// TIA Portal V18 export
// export: Created 2026-06-08T16:32:21.3339851Z, ExportSetting WithDefaults, DisplayName Totally Integrated Automation Portal, DisplayVersion V18, DisplayName TIA Portal Openness, DisplayVersion V18, DisplayName TIA Portal Version Control Interface, DisplayVersion V18, DisplayName STEP 7 Professional, DisplayVersion V18, DisplayName STEP 7 Safety, DisplayVersion V18, DisplayName WinCC Professional, DisplayVersion V18
FUNCTION_BLOCK "Assembly_conv"   // FB9, LAD
VERSION : 0.1
// stored: AutoNumber true, IsIECCheckEnabled false, UDAEnableTagReadback false
   VAR_TEMP   // added for the SCL form of the ladder/FBD networks
      _w1 : Bool;
      _s5time1 : S5Time;
   END_VAR
BEGIN

REGION Network 1
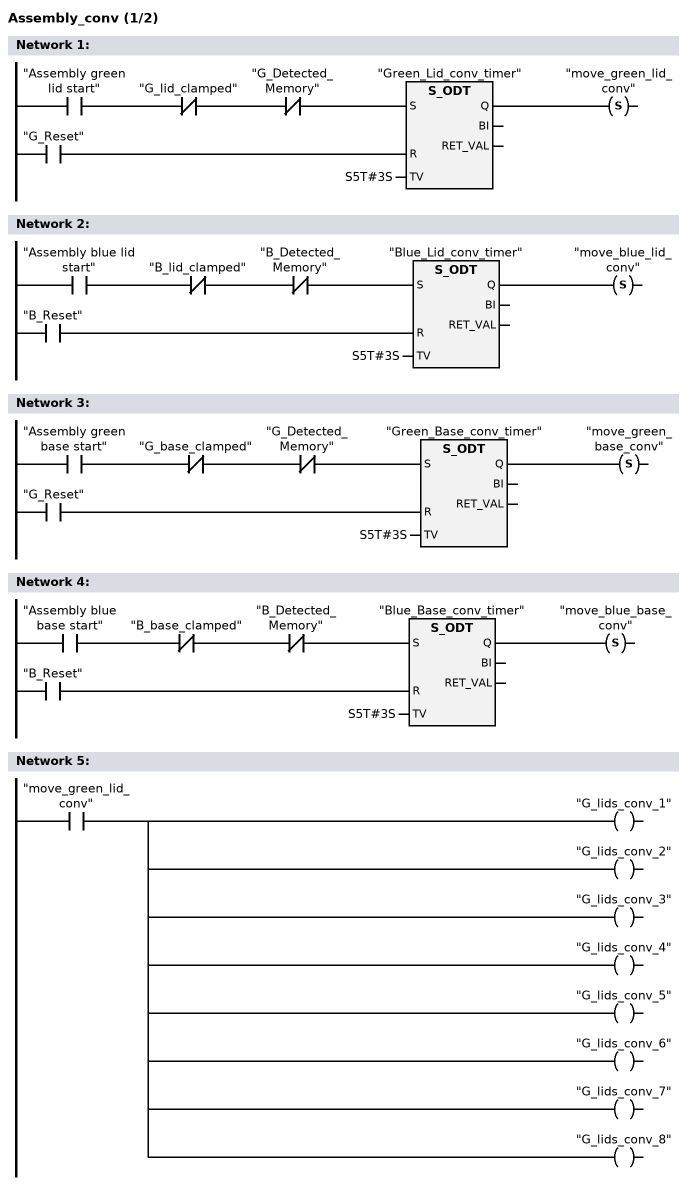
   RUNG wire#powerrail
      Contact( "Assembly green lid start" )
      I_Contact( "G_lid_clamped" )
      I_Contact( "G_Detected_Memory" )
      S_ODT(T_NO := "Green_Lid_conv_timer", R := wire#w1, TV := S5T#3S, BI =>, RET_VAL =>)
      S_Coil( "move_green_lid_conv" )
   END_RUNG
   RUNG wire#powerrail
      Contact( "G_Reset" )
   END_RUNG wire#w1
   // the same network as SCL:
   #_s5time1 := S_ODT(T_NO := "Green_Lid_conv_timer",
                      S := "Assembly green lid start" AND NOT "G_lid_clamped" AND NOT "G_Detected_Memory",
                      R := "G_Reset",
                      TV := S5T#3S,
                      Q => #_w1);
   IF #_w1 THEN "move_green_lid_conv" := TRUE; END_IF;
END_REGION

REGION Network 2
   RUNG wire#powerrail
      Contact( "Assembly blue lid start" )
      I_Contact( "B_lid_clamped" )
      I_Contact( "B_Detected_Memory" )
      S_ODT(T_NO := "Blue_Lid_conv_timer", R := wire#w1, TV := S5T#3S, BI =>, RET_VAL =>)
      S_Coil( "move_blue_lid_conv" )
   END_RUNG
   RUNG wire#powerrail
      Contact( "B_Reset" )
   END_RUNG wire#w1
   // the same network as SCL:
   #_s5time1 := S_ODT(T_NO := "Blue_Lid_conv_timer",
                      S := "Assembly blue lid start" AND NOT "B_lid_clamped" AND NOT "B_Detected_Memory",
                      R := "B_Reset",
                      TV := S5T#3S,
                      Q => #_w1);
   IF #_w1 THEN "move_blue_lid_conv" := TRUE; END_IF;
END_REGION

REGION Network 3
   RUNG wire#powerrail
      Contact( "Assembly green base start" )
      I_Contact( "G_base_clamped" )
      I_Contact( "G_Detected_Memory" )
      S_ODT(T_NO := "Green_Base_conv_timer", R := wire#w1, TV := S5T#3S, BI =>, RET_VAL =>)
      S_Coil( "move_green_base_conv" )
   END_RUNG
   RUNG wire#powerrail
      Contact( "G_Reset" )
   END_RUNG wire#w1
   // the same network as SCL:
   #_s5time1 := S_ODT(T_NO := "Green_Base_conv_timer",
                      S := "Assembly green base start" AND NOT "G_base_clamped" AND NOT "G_Detected_Memory",
                      R := "G_Reset",
                      TV := S5T#3S,
                      Q => #_w1);
   IF #_w1 THEN "move_green_base_conv" := TRUE; END_IF;
END_REGION

REGION Network 4
   RUNG wire#powerrail
      Contact( "Assembly blue base start" )
      I_Contact( "B_base_clamped" )
      I_Contact( "B_Detected_Memory" )
      S_ODT(T_NO := "Blue_Base_conv_timer", R := wire#w1, TV := S5T#3S, BI =>, RET_VAL =>)
      S_Coil( "move_blue_base_conv" )
   END_RUNG
   RUNG wire#powerrail
      Contact( "B_Reset" )
   END_RUNG wire#w1
   // the same network as SCL:
   #_s5time1 := S_ODT(T_NO := "Blue_Base_conv_timer",
                      S := "Assembly blue base start" AND NOT "B_base_clamped" AND NOT "B_Detected_Memory",
                      R := "B_Reset",
                      TV := S5T#3S,
                      Q => #_w1);
   IF #_w1 THEN "move_blue_base_conv" := TRUE; END_IF;
END_REGION

REGION Network 5
   RUNG wire#powerrail
      Contact( "move_green_lid_conv" )
      wire#w1
      Coil( "G_lids_conv_1" )
   END_RUNG
   RUNG wire#w1
      Coil( "G_lids_conv_2" )
   END_RUNG
   RUNG wire#w1
      Coil( "G_lids_conv_3" )
   END_RUNG
   RUNG wire#w1
      Coil( "G_lids_conv_4" )
   END_RUNG
   RUNG wire#w1
      Coil( "G_lids_conv_5" )
   END_RUNG
   RUNG wire#w1
      Coil( "G_lids_conv_6" )
   END_RUNG
   RUNG wire#w1
      Coil( "G_lids_conv_7" )
   END_RUNG
   RUNG wire#w1
      Coil( "G_lids_conv_8" )
   END_RUNG
   // the same network as SCL:
   "G_lids_conv_1" := "move_green_lid_conv";
   "G_lids_conv_2" := "move_green_lid_conv";
   "G_lids_conv_3" := "move_green_lid_conv";
   "G_lids_conv_4" := "move_green_lid_conv";
   "G_lids_conv_5" := "move_green_lid_conv";
   "G_lids_conv_6" := "move_green_lid_conv";
   "G_lids_conv_7" := "move_green_lid_conv";
   "G_lids_conv_8" := "move_green_lid_conv";
END_REGION

REGION Network 6
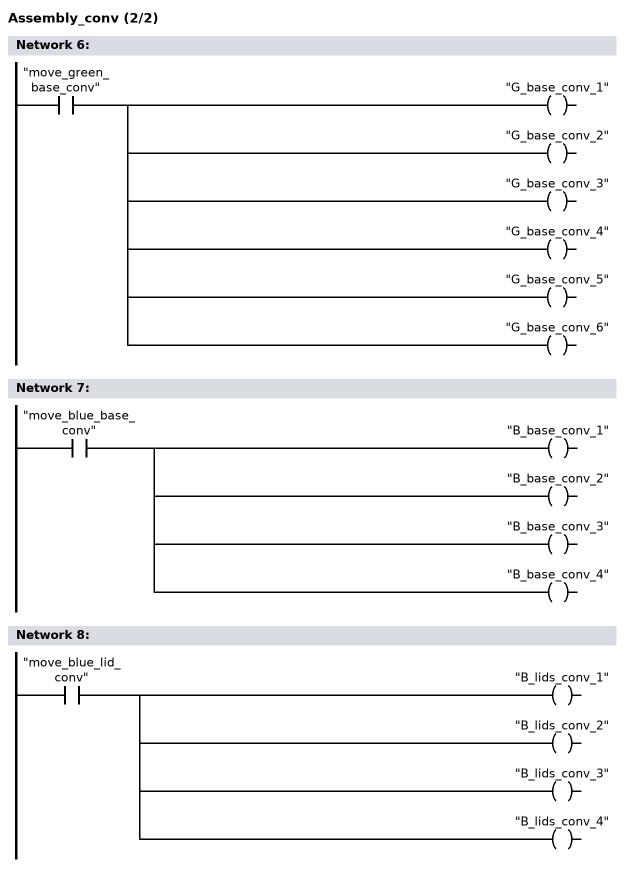
   RUNG wire#powerrail
      Contact( "move_green_base_conv" )
      wire#w1
      Coil( "G_base_conv_1" )
   END_RUNG
   RUNG wire#w1
      Coil( "G_base_conv_2" )
   END_RUNG
   RUNG wire#w1
      Coil( "G_base_conv_3" )
   END_RUNG
   RUNG wire#w1
      Coil( "G_base_conv_4" )
   END_RUNG
   RUNG wire#w1
      Coil( "G_base_conv_5" )
   END_RUNG
   RUNG wire#w1
      Coil( "G_base_conv_6" )
   END_RUNG
   // the same network as SCL:
   "G_base_conv_1" := "move_green_base_conv";
   "G_base_conv_2" := "move_green_base_conv";
   "G_base_conv_3" := "move_green_base_conv";
   "G_base_conv_4" := "move_green_base_conv";
   "G_base_conv_5" := "move_green_base_conv";
   "G_base_conv_6" := "move_green_base_conv";
END_REGION

REGION Network 7
   RUNG wire#powerrail
      Contact( "move_blue_base_conv" )
      wire#w1
      Coil( "B_base_conv_1" )
   END_RUNG
   RUNG wire#w1
      Coil( "B_base_conv_2" )
   END_RUNG
   RUNG wire#w1
      Coil( "B_base_conv_3" )
   END_RUNG
   RUNG wire#w1
      Coil( "B_base_conv_4" )
   END_RUNG
   // the same network as SCL:
   "B_base_conv_1" := "move_blue_base_conv";
   "B_base_conv_2" := "move_blue_base_conv";
   "B_base_conv_3" := "move_blue_base_conv";
   "B_base_conv_4" := "move_blue_base_conv";
END_REGION

REGION Network 8
   RUNG wire#powerrail
      Contact( "move_blue_lid_conv" )
      wire#w1
      Coil( "B_lids_conv_1" )
   END_RUNG
   RUNG wire#w1
      Coil( "B_lids_conv_2" )
   END_RUNG
   RUNG wire#w1
      Coil( "B_lids_conv_3" )
   END_RUNG
   RUNG wire#w1
      Coil( "B_lids_conv_4" )
   END_RUNG
   // the same network as SCL:
   "B_lids_conv_1" := "move_blue_lid_conv";
   "B_lids_conv_2" := "move_blue_lid_conv";
   "B_lids_conv_3" := "move_blue_lid_conv";
   "B_lids_conv_4" := "move_blue_lid_conv";
END_REGION
END_FUNCTION_BLOCK
